TYPE E_WinchMode :
(
    Off := 0,
    Manual := 1,
    Auto := 2
);
END_TYPE

(* stored: Version 1.1.0.1
   DUT DUT_WinchMode: Id {a96df46c-1192-4a89-a363-ec7b37544f8f} *)
